Staubli VAL3: interfaceDefault.pjx

--- interfaceDefault.pjx ---
Parameters version=s7.11 stackSize=5000 millimeterUnit=true
Program file=ack.pgx
Program file=clearScreen.pgx
Program file=debug.pgx
Program file=feedbackStatus.pgx
Program file=init.pgx
Program file=motionBuffer.pgx
Program file=motionProgress.pgx
Program file=motionStatus.pgx
Program file=start.pgx
Program file=stop.pgx
Program file=trajBuffer.pgx
Program file=velOverwrite.pgx
Data file=interfaceDefault.dtx
Library alias=libQueueFuncs path=Disk://ros_libs/QueueFuncs/QueueFuncs.pjx

--- cartStatus.pgx ---
public program cartStatus(num x_nCartConnFlag, num x_nLastMsgAge)
begin

  // Do nothing
  // See start() program for more details

end
